// TIA Portal project "AspenFormation" (V17)

(* hardware
DEVICE "S7-1200 station_2"  S7-1200 Station
   slot 0: "Rack_0"  S7-1200 Rack  Rack  V1.0
   slot 1: "PLC_2"  CPU 1215C AC/DC/Rly  6ES7 215-1BG31-0XB0  V3.0
   slot 3: "AQ 1x12BIT_1"  AQ1 signal board  6ES7 232-4HA30-0XB0  V1.0
   slot 101: "CM 1241 (RS485)_1"  CM 1241 (RS485)  6ES7 241-1CH30-0XB0  V1.0
*)

// ===== PLC "PLC_2"  CPU 1215C AC/DC/Rly =====

VAR_GLOBAL   // PLC tag table "Default tag table"
   "Tag_1" AT %I0.0 : Bool;
   "Tag_3" AT %I0.1 : Bool;
   "Tag_5" AT %I0.2 : Bool;
   "Tag_6" AT %I0.3 : Bool;
   "Tag_8" AT %I0.4 : Bool;
   "Tag_2" AT %Q0.1 : Bool;
   "Tag_4" AT %Q0.2 : Bool;
   "Tag_7" AT %Q0.3 : Bool;
   "Start" AT %M0.0 : Bool;
   "Pression" AT %MW10 : Int;
   "temp" AT %MD12 : Real;
   "temps" AT %MD16 : Time;
   "moteur1" AT %MD20 : Time;
   "System_Byte" AT %MB1 : Byte;
   "FirstScan" AT %M1.0 : Bool;
   "DiagStatusUpdate" AT %M1.1 : Bool;
   "AlwaysTRUE" AT %M1.2 : Bool;
   "AlwaysFALSE" AT %M1.3 : Bool;
   "Clock_Byte" AT %MB0 : Byte;
   "Clock_10Hz" AT %M0.0 : Bool;
   "Clock_5Hz" AT %M0.1 : Bool;
   "Clock_2.5Hz" AT %M0.2 : Bool;
   "Clock_2Hz" AT %M0.3 : Bool;
   "Clock_1.25Hz" AT %M0.4 : Bool;
   "Clock_1Hz" AT %M0.5 : Bool;
   "Clock_0.625Hz" AT %M0.6 : Bool;
   "Clock_0.5Hz" AT %M0.7 : Bool;
END_VAR

TYPE "User_data_type_1"
VERSION : 0.1
   STRUCT
      CommandeMoteur : Struct
         cmda : Bool;
         cmdar : Bool;
      END_STRUCT;
   END_STRUCT;
END_TYPE

DATA_BLOCK "MON_FB_DB"   // DB1
{ S7_Optimized_Access := 'TRUE' }
VERSION : 0.1
// stored: InstanceOfName MON_FB
"MON_FB"
BEGIN
END_DATA_BLOCK

DATA_BLOCK "Donne"   // DB2
{ S7_Optimized_Access := 'FALSE' }
VERSION : 0.1
   VAR
      var1 : Bool;
      var2 : Bool;
      int1 : DInt := 200;
      int2 : Int;
   END_VAR
BEGIN
END_DATA_BLOCK

FUNCTION_BLOCK "MON_FB"   // FB1, LAD
{ S7_Optimized_Access := 'TRUE' }
VERSION : 0.1
BEGIN

REGION Network 1
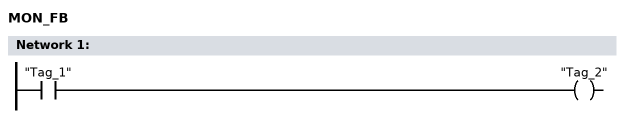
   RUNG wire#powerrail
      Contact( "Tag_1" )
      Coil( "Tag_2" )
   END_RUNG
   // the same network as SCL:
   "Tag_2" := "Tag_1";
END_REGION

REGION Network 2 (SCL)
   IF "Tag_3" THEN
       // Statement section IF
       "Tag_4" := TRUE;
   ELSE
       "Tag_4" := FALSE;
   END_IF;
END_REGION
END_FUNCTION_BLOCK

FUNCTION "Block_1" : Void   // FC1, LAD
{ S7_Optimized_Access := 'TRUE' }
VERSION : 0.1
   VAR_INPUT
      input1 : Bool;
      input2 : Bool;
   END_VAR
   VAR_OUTPUT
      output : Bool;
      ouput2 : Bool;
   END_VAR
   VAR_IN_OUT
      inoutput : Bool;
   END_VAR
BEGIN

REGION Network 1
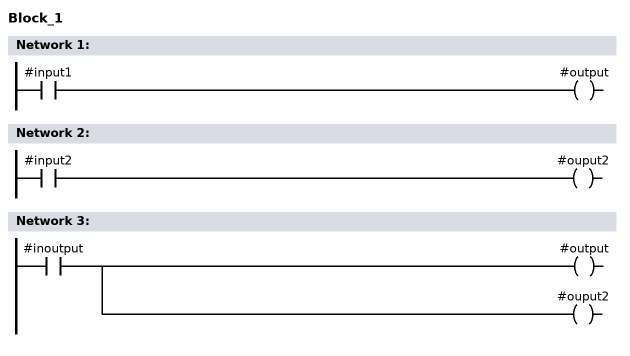
   RUNG wire#powerrail
      Contact( #input1 )
      Coil( #output )
   END_RUNG
   // the same network as SCL:
   #output := #input1;
END_REGION

REGION Network 2
   RUNG wire#powerrail
      Contact( #input2 )
      Coil( #ouput2 )
   END_RUNG
   // the same network as SCL:
   #ouput2 := #input2;
END_REGION

REGION Network 3
   RUNG wire#powerrail
      Contact( #inoutput )
      wire#w1
      Coil( #output )
   END_RUNG
   RUNG wire#w1
      Coil( #ouput2 )
   END_RUNG
   // the same network as SCL:
   #output := #inoutput;
   #ouput2 := #inoutput;
END_REGION
END_FUNCTION

ORGANIZATION_BLOCK "Main"   // OB1, LAD, ProgramCycle
TITLE = "Main Program Sweep (Cycle)"
{ S7_Optimized_Access := 'TRUE' }
VERSION : 0.1
BEGIN

REGION Network 1
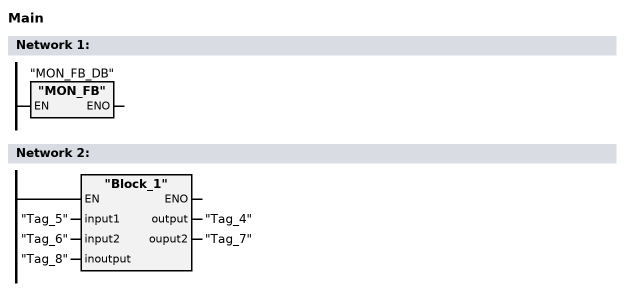
   RUNG wire#powerrail
      "MON_FB_DB"()
   END_RUNG
   // the same network as SCL:
   "MON_FB_DB"();   // "MON_FB"
END_REGION

REGION Network 2
   RUNG wire#powerrail
      "Block_1"(input1 := "Tag_5", input2 := "Tag_6", inoutput := "Tag_8", output => "Tag_4", ouput2 => "Tag_7")
   END_RUNG
   // the same network as SCL:
   "Block_1"(input1 := "Tag_5", input2 := "Tag_6", inoutput := "Tag_8", output => "Tag_4", ouput2 => "Tag_7");
END_REGION
END_ORGANIZATION_BLOCK

ORGANIZATION_BLOCK "Startup"   // OB100, LAD, Startup
TITLE = "Complete Restart"
{ S7_Optimized_Access := 'TRUE' }
VERSION : 0.1
   VAR_INPUT
      LostRetentive : Bool;   // True if retentive data are lost
      LostRTC : Bool;   // True if date and time are lost
   END_VAR
BEGIN
END_ORGANIZATION_BLOCK